(* CODESYS project mixer process control.project

Project tree, tasks and I/O mapping:
  Device : CODESYS Control Win V3, 3S - Smart Software Solutions GmbH, order no. 305021, version 3.5.7.0
    application Application
      libraries: Standard, * (System)
      task MainTask (cyclic, interval t#20ms, priority 1) calls PLC_PRG
      task VISU_TASK (cyclic, interval 100 ms, priority 31) calls VisuElems.Visu_Prg
      program PLC_PRG [LD]
      visualisation Visualization
  text list GlobalTextList
*)

// Device/Application/PLC_PRG
PROGRAM PLC_PRG
VAR
	start: BOOL;
	stop: BOOL;
	process_on: BOOL;
	prsw: BOOL;
	tpsw: BOOL;
	pb: BOOL;
	m: BOOL;
END_VAR

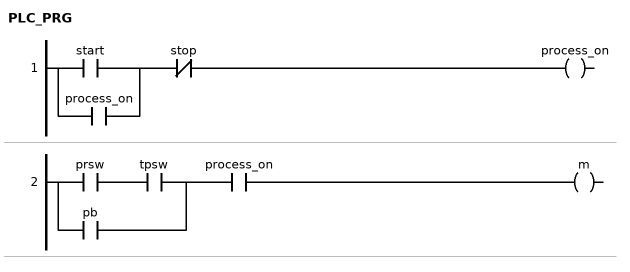
// NETWORK 1
process_on := (start OR process_on) AND NOT stop;

// NETWORK 2
m := (prsw AND tpsw OR pb) AND process_on;

END_PROGRAM

// Device/Application/Visualization
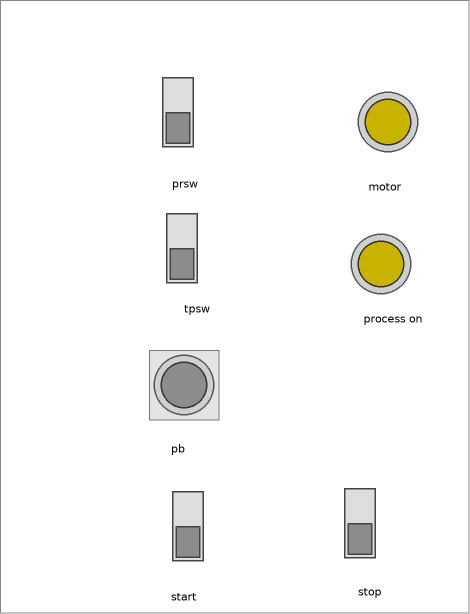
VISUALIZATION Visualization  // 470x614
    DipSwitch (143,77 70x70), variable: PLC_PRG.prsw, behaviour: TOGGLE, style: Switch-DipSwitch-Gray
    DipSwitch (147,213 70x70), variable: PLC_PRG.tpsw, behaviour: TOGGLE, style: Switch-DipSwitch-Gray
    DipSwitch (153,491 70x70), variable: PLC_PRG.start, behaviour: TOGGLE, style: Switch-DipSwitch-Gray
    DipSwitch (325,488 70x70), variable: PLC_PRG.stop, behaviour: TOGGLE, style: Switch-DipSwitch-Gray
    PushSwitch (149,350 70x70), variable: PLC_PRG.pb, behaviour: TOGGLE, style: Switch-PushSwitch-Gray
    Lamp1 (353,87 70x70), variable: PLC_PRG.m, style: Lamp-Lamp1-Yellow
    Lamp1 (346,229 70x70), variable: PLC_PRG.process_on, style: Lamp-Lamp1-Yellow
    Label (110,169 150x30), "prsw"
    Label (310,172 150x30), "motor"
    Label (122,294 150x30), "tpsw"
    Label (318,304 150x30), "process on"
    Label (103,434 150x30), "pb"
    Label (109,582 150x30), "start"
    Label (295,577 150x30), "stop"
END_VISUALIZATION
